{attribute 'GeneratedUsingTerminal: EL2262--0000'}
{attribute addProperty BoxType "EL2262--0000"}
{attribute addProperty Id "EtcSlaveTerminalBaseCycle_CounterAT %Q*Cycle_Counter_2C2338042Sample_0AT %Q*Sample_3C4603C71WcStateAT %I*WcState_0B2B16F91InfoDataAT %I*InfoData_A7436BC610"}
{attribute addProperty CRC "3996278071"}
{attribute addProperty Size "14"}
TYPE EL2262_EE325D37 EXTENDS EtcSlaveTerminalBase :
STRUCT
	{attribute addProperty Name "Cycle_Counter"}
	Cycle_Counter : Cycle_Counter_2C233804;
	{attribute addProperty Name "Sample_0"}
	Sample_0 : Sample_3C4603C7;
	{attribute addProperty Name "WcState"}
	WcState : WcState_0B2B16F9;
	{attribute addProperty Name "InfoData"}
	InfoData : InfoData_A7436BC6;
END_STRUCT
END_TYPE

(* stored: Version 1.2.0.0, ProductVersion 3.1.4024.9
   DUT EL2262_EE325D37: Id {d7ca0de9-94a3-4f14-9799-7e0a5b717b00} *)
